INTERFACE ITF_pompangout

METHOD set : INT
VAR_INPUT
		state : INT;
END_VAR
END_METHOD

END_INTERFACE

(* stored: Version 1.1.0.1, ProductVersion 3.1.4026.8
   Itf ITF_pompangout: Id {7533d3ce-6466-4061-80e4-d53d50a1fdea}
   Method set: Id {f6786b9e-2847-416b-bb68-baf54047f394} *)
